{attribute 'qualified_only'}
{attribute 'strict'}
TYPE E_AirpadBrake :
(
    eStandard := 0,
    eAirpad := 1,
    eExternalBrake := 2
):=eStandard;
END_TYPE

(* stored: Version 1.1.0.1
   DUT E_AirpadBrake: Id {6960b210-0ca5-0601-1372-7c299d82f9b8} *)
